Staubli VAL3: TrajByPass.pgx

public program TrajByPass(num x_nIndex, num x_nTotal)
begin


 // 路径由外部信号过滤
 // 实现方式
 //通过一个数字量输入信号，一个模拟量输入信号，一个模拟量输出信号
 //没有经过测试过



  do

    call IO:TrajBypass(TxtFile:bBypass[x_nIndex-1],x_nIndex-1)
    x_nIndex=x_nIndex+1
    delay(0)
  until TxtFile:bBypass[x_nIndex-1]==false or x_nIndex>=x_nTotal



end
